Staubli VAL3: setTool.pgx

public program setTool(string x_sTool)
begin
  //
  sToolName=x_sTool
end
